FUNCTION_BLOCK FB_LeakDetection

VAR
	bValveOpen : BOOL;
	bFlowSensor : BOOL;
	
	fbTon : TON;
	fbTp : TP;
	
	bAlarm : BOOL;
	tFlowTime : TIME := T#2S;
	tAlarmDuration : TIME := T#5S;
END_VAR

fbTon(IN := bValveOpen , PT := tFlowTime);
IF fbTon.Q THEN
	bFlowSensor := TRUE;
ELSE
	bFlowSensor := FALSE;
END_IF

fbTp(IN := bFlowSensor,PT := tAlarmDuration);
bAlarm := fbTp.Q;

END_FUNCTION_BLOCK

(* stored: Version 1.1.0.1, ProductVersion 3.1.4024.16
   POU FB_LeakDetection: Id {dfc3e555-b056-4447-b785-158c973fb351}, SpecialFunc None *)
